ABB RAPID module: Project.mod

MODULE MainModule
    TASK PERS tooldata tool1:=[TRUE,[[3.25653,-2.2499,106.27],[1,0,0,0]],[0.2,[0,0,50],[1,0,0,0],0,0,0]];
    VAR robtarget p_home := [[342.30,-38.16,327.52],[1.20614E-05,0.456804,-0.889567,-5.42704E-06],[-1,-1,-1,0],[9E+09,9E+09,9E+09,9E+09,9E+09,9E+09]];

    VAR robtarget p_home := [[342.30,-38.16,327.52],[1.20614E-05,0.456804,-0.889567,-5.42704E-06],[-1,-1,-1,0],[9E+09,9E+09,9E+09,9E+09,9E+09,9E+09]];
    VAR robtarget p_home := [[342.30,-38.16,327.52],[1.20614E-05,0.456804,-0.889567,-5.42704E-06],[-1,-1,-1,0],[9E+09,9E+09,9E+09,9E+09,9E+09,9E+09]];
    VAR robtarget p_home := [[342.30,-38.16,327.52],[1.20614E-05,0.456804,-0.889567,-5.42704E-06],[-1,-1,-1,0],[9E+09,9E+09,9E+09,9E+09,9E+09,9E+09]];
    VAR robtarget p_home := [[342.30,-38.16,327.52],[1.20614E-05,0.456804,-0.889567,-5.42704E-06],[-1,-1,-1,0],[9E+09,9E+09,9E+09,9E+09,9E+09,9E+09]];
    VAR robtarget p_home := [[342.30,-38.16,327.52],[1.20614E-05,0.456804,-0.889567,-5.42704E-06],[-1,-1,-1,0],[9E+09,9E+09,9E+09,9E+09,9E+09,9E+09]];
    VAR robtarget p_home := [[342.30,-38.16,327.52],[1.20614E-05,0.456804,-0.889567,-5.42704E-06],[-1,-1,-1,0],[9E+09,9E+09,9E+09,9E+09,9E+09,9E+09]];
    VAR robtarget p_home := [[342.30,-38.16,327.52],[1.20614E-05,0.456804,-0.889567,-5.42704E-06],[-1,-1,-1,0],[9E+09,9E+09,9E+09,9E+09,9E+09,9E+09]];
    VAR robtarget p_home := [[342.30,-38.16,327.52],[1.20614E-05,0.456804,-0.889567,-5.42704E-06],[-1,-1,-1,0],[9E+09,9E+09,9E+09,9E+09,9E+09,9E+09]];
    VAR robtarget p_home := [[342.30,-38.16,327.52],[1.20614E-05,0.456804,-0.889567,-5.42704E-06],[-1,-1,-1,0],[9E+09,9E+09,9E+09,9E+09,9E+09,9E+09]];
    VAR robtarget p_home := [[342.30,-38.16,327.52],[1.20614E-05,0.456804,-0.889567,-5.42704E-06],[-1,-1,-1,0],[9E+09,9E+09,9E+09,9E+09,9E+09,9E+09]];
    VAR robtarget p_home := [[342.30,-38.16,327.52],[1.20614E-05,0.456804,-0.889567,-5.42704E-06],[-1,-1,-1,0],[9E+09,9E+09,9E+09,9E+09,9E+09,9E+09]];
    VAR robtarget p_home := [[342.30,-38.16,327.52],[1.20614E-05,0.456804,-0.889567,-5.42704E-06],[-1,-1,-1,0],[9E+09,9E+09,9E+09,9E+09,9E+09,9E+09]];
    VAR robtarget p_home := [[342.30,-38.16,327.52],[1.20614E-05,0.456804,-0.889567,-5.42704E-06],[-1,-1,-1,0],[9E+09,9E+09,9E+09,9E+09,9E+09,9E+09]];
    VAR robtarget p_home := [[342.30,-38.16,327.52],[1.20614E-05,0.456804,-0.889567,-5.42704E-06],[-1,-1,-1,0],[9E+09,9E+09,9E+09,9E+09,9E+09,9E+09]];
    VAR robtarget p_home := [[342.30,-38.16,327.52],[1.20614E-05,0.456804,-0.889567,-5.42704E-06],[-1,-1,-1,0],[9E+09,9E+09,9E+09,9E+09,9E+09,9E+09]];
    VAR robtarget p_home := [[342.30,-38.16,327.52],[1.20614E-05,0.456804,-0.889567,-5.42704E-06],[-1,-1,-1,0],[9E+09,9E+09,9E+09,9E+09,9E+09,9E+09]];
    VAR robtarget p_home := [[342.30,-38.16,327.52],[1.20614E-05,0.456804,-0.889567,-5.42704E-06],[-1,-1,-1,0],[9E+09,9E+09,9E+09,9E+09,9E+09,9E+09]];
    VAR robtarget p_home := [[342.30,-38.16,327.52],[1.20614E-05,0.456804,-0.889567,-5.42704E-06],[-1,-1,-1,0],[9E+09,9E+09,9E+09,9E+09,9E+09,9E+09]];


ENDMODULE
